(* IEC 61131-3 sources: test_training/GmpAccess2/src/Variables, 1 file *)

(* ---- GlobalVariables.gvl ---- *)
VAR_GLOBAL
	gSetState 		: STRING := 'SIMULATION'; (* state can be switched *)
	triggerScope 	: BOOL;
	exportScope 	: BOOL;
	scopeState 		: GMP232X_SCOPE_STATE;
END_VAR

VAR_GLOBAL CONSTANT
	MODULE_NUMBER 	: INT := 24;
END_VAR
